(* IEC 61131-3 sources: AXOpen/src/showcase/app/src/components.abb.robotics/Documentation, 3 files *)

(* ---- AbbRobotics.st ---- *)
USING AXOpen.Core;
NAMESPACE AXOpen.Components.Abb.Robotics
    {S7.extern=ReadWrite}
    CLASS AbbRobotics EXTENDS AXOpen.Core.AxoObject
        VAR PUBLIC
            _rootObject  : AxoObject;
            axoIrc5_v_1_x_x : AxoIrc5_v_1_x_x_Showcase;
            axoOmnicore_v_1_x_x : AxoOmnicore_v_1_x_x_Showcase;
        END_VAR

        METHOD PUBLIC Execute
            _rootObject.Run(THIS);
            axoIrc5_v_1_x_x.Run(_rootObject);
            axoOmnicore_v_1_x_x.Run(_rootObject);
        END_METHOD
    END_CLASS
END_NAMESPACE

(* ---- AxoIrc5_v_1_x_x_Showcase.st ---- *)
USING AXOpen.Core;
NAMESPACE AXOpen.Components.Abb.Robotics
    {S7.extern=ReadWrite}
    CLASS AxoIrc5_v_1_x_x_Showcase EXTENDS AXOpen.Core.AxoObject
        //<ComponentDeclaration>
        VAR PUBLIC
            AxoIrc5_v_1_x_x : AXOpen.Components.Abb.Robotics.AxoIrc5_v_1_x_x;
        END_VAR
        //</ComponentDeclaration>

        //<InitializationArgumentsDeclaration>
        VAR PUBLIC
            movementParams : AXOpen.Components.Abstractions.Robotics.AxoRoboticsMovementsParams;
            manualControl   :   BOOL;
        END_VAR
        //</InitializationArgumentsDeclaration>

        METHOD PUBLIC OVERRIDE Run
            VAR_INPUT
                inParent : IAxoObject;
            END_VAR
            SUPER.Run(inParent);

            IF(manualControl) THEN
                AxoIrc5_v_1_x_x.ActivateManualControl();
            END_IF;

            //<Initialization>
            AxoIrc5_v_1_x_x.Run(inParent          := inParent,
                                hwID            :=  AXOpen.Showcase.HwIdentifiers#abb_irc5_robot_HwID);
            //</Initialization>

            THIS.UseInSequencer();
        END_METHOD

        //<Usage>
        VAR PUBLIC
            Sequencer : AxoSequencer;
            Steps : ARRAY[0..18] OF AXOpen.Core.AxoStep;
        END_VAR

        METHOD PRIVATE UseInSequencer

            Sequencer.Run(THIS);
            Sequencer.Open();
            Sequencer.SequenceMode := eAxoSequenceMode#RunOnce;

            IF(Steps[0].Execute(Sequencer, 'Restore')) THEN
                manualControl := FALSE;
                AxoIrc5_v_1_x_x.Config.InfoTime      := LTIME#2S;
                AxoIrc5_v_1_x_x.Config.TaskTimeout   := LTIME#0S;
                AxoIrc5_v_1_x_x.Config.ErrorTime     := LTIME#0S;
                AxoIrc5_v_1_x_x.Restore();
                Sequencer.MoveNext();
            END_IF;

            IF(Steps[1].Execute(Sequencer, 'Start at main')) THEN
                IF(AxoIrc5_v_1_x_x.StartAtMain().IsDone()) THEN
                    Sequencer.MoveNext();
                END_IF;
            END_IF;

            IF(Steps[2].Execute(Sequencer, 'Start motors and program')) THEN
                IF(AxoIrc5_v_1_x_x.StartMotorsAndProgram().IsDone()) THEN
                    Sequencer.MoveNext();
                END_IF;
            END_IF;

            IF(Steps[3].Execute(Sequencer, 'Move to position 100')) THEN
                movementParams.ActionNo         :=  BYTE#100;
                movementParams.GlobalSpeed      :=  BYTE#5;
                movementParams.ToolNo           :=  BYTE#10;
                movementParams.WorkobjectNo     :=  BYTE#15;
                movementParams.PointNo          :=  BYTE#20;
                movementParams.UserSpecSpeed1   :=  INT#25;
                movementParams.UserSpecSpeed2   :=  INT#30;
                movementParams.Coordinates.X    :=  REAL#1.2;
                movementParams.Coordinates.Y    :=  REAL#2.3;
                movementParams.Coordinates.Z    :=  REAL#3.4;
                movementParams.Coordinates.Rx   :=  REAL#4.5;
                movementParams.Coordinates.Ry   :=  REAL#5.6;
                movementParams.Coordinates.Rz   :=  REAL#6.7;

                IF(AxoIrc5_v_1_x_x.StartMovements(movementParams).IsDone()) THEN
                    AxoIrc5_v_1_x_x.StartMovementsTask.Restore();
                    Sequencer.MoveNext();
                END_IF;
            END_IF;

            IF(Steps[4].Execute(Sequencer, 'Move to position 1')) THEN
                movementParams.ActionNo             :=  BYTE#1;

                IF(AxoIrc5_v_1_x_x.StartMovements(movementParams).IsDone()) THEN
                    AxoIrc5_v_1_x_x.StartMovementsTask.Restore();
                    Sequencer.MoveNext();
                END_IF;
            END_IF;

            IF(Steps[5].Execute(Sequencer, 'Move to position 3')) THEN
                movementParams.ActionNo             :=  BYTE#3;

                IF(AxoIrc5_v_1_x_x.StartMovements(movementParams).IsBusy() AND Sequencer.CurrentStep.Duration >= T#500ms) THEN
                    Sequencer.MoveNext();
                END_IF;
            END_IF;
            // Simulation of the entering the robotic cell during movement =>
            IF(Steps[6].Execute(Sequencer, 'Stop during movement')) THEN
                AxoIrc5_v_1_x_x.StartMovements(movementParams); // <- This line just emulates the cyclical call of the movement method
                IF(AxoIrc5_v_1_x_x.StopMovements().IsDone()) THEN
                    Sequencer.MoveNext();
                END_IF;
            END_IF;

            IF(Steps[7].Execute(Sequencer, '<#Unlocking and opening the robotic cell#>')) THEN
                //-------------------------------------------------------
                AxoIrc5_v_1_x_x.StartMovements(movementParams); // <- This line just emulates the cyclical call of the movement method
                IF (TRUE) THEN
                    Sequencer.MoveNext();
                END_IF;
                //-------------------------------------------------------
            END_IF;

            IF (Steps[8].Execute(Sequencer, '<#Closing and locking the robotic cell#>')) THEN
                //-------------------------------------------------------
                AxoIrc5_v_1_x_x.StartMovements(movementParams); // <- This line just emulates the cyclical call of the movement method
                IF (TRUE) THEN
                    Sequencer.MoveNext();
                END_IF;
                //-------------------------------------------------------
            END_IF;
            // <= Simulation of the entering the robotic cell during movement

            IF(Steps[9].Execute(Sequencer, 'Start motors and program')) THEN
                AxoIrc5_v_1_x_x.StartMovements(movementParams); // <- This line just emulates the cyclical call of the movement method
                IF(AxoIrc5_v_1_x_x.StartMotorsAndProgram().IsDone()) THEN // <- Starting motor and program after safety circuit has been interupted
                    Sequencer.MoveNext();
                END_IF;
            END_IF;

            IF(Steps[10].Execute(Sequencer, 'Continue to position 3')) THEN
                IF(AxoIrc5_v_1_x_x.StartMovementsTask.IsDone()) THEN
                    AxoIrc5_v_1_x_x.StartMovementsTask.Restore();
                    Sequencer.MoveNext();
                END_IF;
            END_IF;

            IF(Steps[11].Execute(Sequencer, 'Move to position 100')) THEN
                movementParams.ActionNo             :=  BYTE#100;

                IF(AxoIrc5_v_1_x_x.StartMovements(movementParams).IsDone()) THEN
                    AxoIrc5_v_1_x_x.StartMovementsTask.Restore();
                    Sequencer.MoveNext();
                END_IF;
            END_IF;

            IF(Steps[12].Execute(Sequencer, 'Move to position 1')) THEN
                movementParams.ActionNo             :=  BYTE#1;

                IF(AxoIrc5_v_1_x_x.StartMovements(movementParams).IsDone()) THEN
                    AxoIrc5_v_1_x_x.StartMovementsTask.Restore();
                    Sequencer.MoveNext();
                END_IF;
            END_IF;

            IF(Steps[13].Execute(Sequencer, 'Stop movement and program')) THEN
                IF(AxoIrc5_v_1_x_x.StopMovementsAndProgram().IsDone()) THEN
                    Sequencer.MoveNext();
                END_IF;
            END_IF;

            IF(Steps[14].Execute(Sequencer, 'Stop motors')) THEN
                IF(AxoIrc5_v_1_x_x.StopMotors().IsDone()) THEN
                    Sequencer.MoveNext();
                END_IF;
            END_IF;

            IF(Steps[15].Execute(Sequencer, 'Start motors, program and movements combined')) THEN
                IF(AxoIrc5_v_1_x_x.StartMotorsProgramAndMovements(movementParams).IsDone()) THEN
                    Sequencer.MoveNext();
                END_IF;
            END_IF;

            IF(Steps[16].Execute(Sequencer, 'Stop program')) THEN
                IF(AxoIrc5_v_1_x_x.StopProgram().IsDone()) THEN
                    Sequencer.MoveNext();
                END_IF;
            END_IF;

            IF(Steps[17].Execute(Sequencer, 'Start program')) THEN
                IF(AxoIrc5_v_1_x_x.StartProgram().IsDone()) THEN
                    Sequencer.MoveNext();
                END_IF;
            END_IF;

            IF(Steps[18].Execute(Sequencer, 'Restore')) THEN
                AxoIrc5_v_1_x_x.Restore();
                Sequencer.CompleteSequence();
            END_IF;
        END_METHOD

        //</Usage>
    END_CLASS
END_NAMESPACE

(* ---- AxoOmnicore_v_1_x_x_Showcase.st ---- *)
USING AXOpen.Core;
NAMESPACE AXOpen.Components.Abb.Robotics
    {S7.extern=ReadWrite}
    CLASS AxoOmnicore_v_1_x_x_Showcase EXTENDS AXOpen.Core.AxoObject
        //<ComponentDeclaration>
        VAR PUBLIC
            AxoOmnicore_v_1_x_x : AXOpen.Components.Abb.Robotics.AxoOmnicore_v_1_x_x;
        END_VAR
        //</ComponentDeclaration>

        //<InitializationArgumentsDeclaration>
        VAR PUBLIC
            movementParams : AXOpen.Components.Abstractions.Robotics.AxoRoboticsMovementsParams;
            manualControl   :   BOOL;
        END_VAR
        //</InitializationArgumentsDeclaration>

        METHOD PUBLIC OVERRIDE Run
            VAR_INPUT
                inParent : IAxoObject;
            END_VAR
            SUPER.Run(inParent);

            IF(manualControl) THEN
                AxoOmnicore_v_1_x_x.ActivateManualControl();
            END_IF;

            //<Initialization>
            AxoOmnicore_v_1_x_x.Run(inParent          := inParent,
                                    hwID            := AXOpen.Showcase.HwIdentifiers#abb_omnicore_robot_HwID);
            //</Initialization>

        THIS.UseInSequencer();
        END_METHOD

        //<Usage>
        VAR PUBLIC
            Sequencer : AxoSequencer;
            Steps : ARRAY[0..18] OF AXOpen.Core.AxoStep;
        END_VAR

        METHOD PRIVATE UseInSequencer

            Sequencer.Run(THIS);
            Sequencer.Open();
            Sequencer.SequenceMode := eAxoSequenceMode#RunOnce;

            IF(Steps[0].Execute(Sequencer, 'Restore')) THEN
                manualControl := FALSE;
                AxoOmnicore_v_1_x_x.Config.InfoTime      := LTIME#2S;
                AxoOmnicore_v_1_x_x.Config.TaskTimeout   := LTIME#0S;
                AxoOmnicore_v_1_x_x.Config.ErrorTime     := LTIME#0S;
                AxoOmnicore_v_1_x_x.Restore();
                Sequencer.MoveNext();
            END_IF;

            IF(Steps[1].Execute(Sequencer, 'Start at main')) THEN
                IF(AxoOmnicore_v_1_x_x.StartAtMain().IsDone()) THEN
                    Sequencer.MoveNext();
                END_IF;
            END_IF;

            IF(Steps[2].Execute(Sequencer, 'Start motors and program')) THEN
                IF(AxoOmnicore_v_1_x_x.StartMotorsAndProgram().IsDone()) THEN
                    Sequencer.MoveNext();
                END_IF;
            END_IF;

            IF(Steps[3].Execute(Sequencer, 'Move to position 100')) THEN
                movementParams.ActionNo         :=  BYTE#100;
                movementParams.GlobalSpeed      :=  BYTE#5;
                movementParams.ToolNo           :=  BYTE#10;
                movementParams.WorkobjectNo     :=  BYTE#15;
                movementParams.PointNo          :=  BYTE#20;
                movementParams.UserSpecSpeed1   :=  INT#25;
                movementParams.UserSpecSpeed2   :=  INT#30;
                movementParams.Coordinates.X    :=  REAL#1.2;
                movementParams.Coordinates.Y    :=  REAL#2.3;
                movementParams.Coordinates.Z    :=  REAL#3.4;
                movementParams.Coordinates.Rx   :=  REAL#4.5;
                movementParams.Coordinates.Ry   :=  REAL#5.6;
                movementParams.Coordinates.Rz   :=  REAL#6.7;

                IF(AxoOmnicore_v_1_x_x.StartMovements(movementParams).IsDone()) THEN
                    AxoOmnicore_v_1_x_x.StartMovementsTask.Restore();
                    Sequencer.MoveNext();
                END_IF;
            END_IF;

            IF(Steps[4].Execute(Sequencer, 'Move to position 1')) THEN
                movementParams.ActionNo             :=  BYTE#1;

                IF(AxoOmnicore_v_1_x_x.StartMovements(movementParams).IsDone()) THEN
                    AxoOmnicore_v_1_x_x.StartMovementsTask.Restore();
                    Sequencer.MoveNext();
                END_IF;
            END_IF;

            IF(Steps[5].Execute(Sequencer, 'Move to position 3')) THEN
                movementParams.ActionNo             :=  BYTE#3;

                IF(AxoOmnicore_v_1_x_x.StartMovements(movementParams).IsBusy() AND Sequencer.CurrentStep.Duration >= T#500ms) THEN
                    Sequencer.MoveNext();
                END_IF;
            END_IF;
            // Simulation of the entering the robotic cell during movement =>
            IF(Steps[6].Execute(Sequencer, 'Stop during movement')) THEN
                AxoOmnicore_v_1_x_x.StartMovements(movementParams); // <- This line just emulates the cyclical call of the movement method
                IF(AxoOmnicore_v_1_x_x.StopMovements().IsDone()) THEN
                    Sequencer.MoveNext();
                END_IF;
            END_IF;

            IF(Steps[7].Execute(Sequencer, '<#Unlocking and opening the robotic cell#>')) THEN
                //-------------------------------------------------------
                AxoOmnicore_v_1_x_x.StartMovements(movementParams); // <- This line just emulates the cyclical call of the movement method
                IF (TRUE) THEN
                    Sequencer.MoveNext();
                END_IF;
                //-------------------------------------------------------
            END_IF;

            IF (Steps[8].Execute(Sequencer, '<#Closing and locking the robotic cell#>')) THEN
                //-------------------------------------------------------
                AxoOmnicore_v_1_x_x.StartMovements(movementParams); // <- This line just emulates the cyclical call of the movement method
                IF (TRUE) THEN
                    Sequencer.MoveNext();
                END_IF;
                //-------------------------------------------------------
            END_IF;
            // <= Simulation of the entering the robotic cell during movement

            IF(Steps[9].Execute(Sequencer, 'Start motors and program')) THEN
                AxoOmnicore_v_1_x_x.StartMovements(movementParams); // <- This line just emulates the cyclical call of the movement method
                IF(AxoOmnicore_v_1_x_x.StartMotorsAndProgram().IsDone()) THEN // <- Starting motor and program after safety circuit has been interupted
                    Sequencer.MoveNext();
                END_IF;
            END_IF;

            IF(Steps[10].Execute(Sequencer, 'Continue to position 3')) THEN
                IF(AxoOmnicore_v_1_x_x.StartMovementsTask.IsDone()) THEN
                    AxoOmnicore_v_1_x_x.StartMovementsTask.Restore();
                    Sequencer.MoveNext();
                END_IF;
            END_IF;

            IF(Steps[11].Execute(Sequencer, 'Move to position 100')) THEN
                movementParams.ActionNo             :=  BYTE#100;

                IF(AxoOmnicore_v_1_x_x.StartMovements(movementParams).IsDone()) THEN
                    AxoOmnicore_v_1_x_x.StartMovementsTask.Restore();
                    Sequencer.MoveNext();
                END_IF;
            END_IF;

            IF(Steps[12].Execute(Sequencer, 'Move to position 1')) THEN
                movementParams.ActionNo             :=  BYTE#1;

                IF(AxoOmnicore_v_1_x_x.StartMovements(movementParams).IsDone()) THEN
                    AxoOmnicore_v_1_x_x.StartMovementsTask.Restore();
                    Sequencer.MoveNext();
                END_IF;
            END_IF;

            IF(Steps[13].Execute(Sequencer, 'Stop movement and program')) THEN
                IF(AxoOmnicore_v_1_x_x.StopMovementsAndProgram().IsDone()) THEN
                    Sequencer.MoveNext();
                END_IF;
            END_IF;

            IF(Steps[14].Execute(Sequencer, 'Stop motors')) THEN
                IF(AxoOmnicore_v_1_x_x.StopMotors().IsDone()) THEN
                    Sequencer.MoveNext();
                END_IF;
            END_IF;

            IF(Steps[15].Execute(Sequencer, 'Start motors, program and movements combined')) THEN
                IF(AxoOmnicore_v_1_x_x.StartMotorsProgramAndMovements(movementParams).IsDone()) THEN
                    Sequencer.MoveNext();
                END_IF;
            END_IF;

            IF(Steps[16].Execute(Sequencer, 'Stop program')) THEN
                IF(AxoOmnicore_v_1_x_x.StopProgram().IsDone()) THEN
                    Sequencer.MoveNext();
                END_IF;
            END_IF;

            IF(Steps[17].Execute(Sequencer, 'Start program')) THEN
                IF(AxoOmnicore_v_1_x_x.StartProgram().IsDone()) THEN
                    Sequencer.MoveNext();
                END_IF;
            END_IF;

            IF(Steps[18].Execute(Sequencer, 'Restore')) THEN
                AxoOmnicore_v_1_x_x.Restore();
                Sequencer.CompleteSequence();
            END_IF;
        END_METHOD

        //</Usage>
    END_CLASS
END_NAMESPACE
